(* LS Electric XG5000 project: PLC_Study *)
(* PLC LSPLC *)
(* module base 0 slot 0: 입력 모듈:XGI-D21A (DC 24V 입력, 8점 (전류소스/싱크입력)) *)
(* module base 0 slot 1: 출력 모듈:XGQ-RY1A (릴레이 출력, 8점 (2A용, 단독 COM.)) *)

(* Comments on direct variables
%QX0.1.0	출력
%QX0.1.2	출력
%IX0.0.3	스위치
*)

PROGRAM NewProgram (* task: 스캔 프로그램 *)

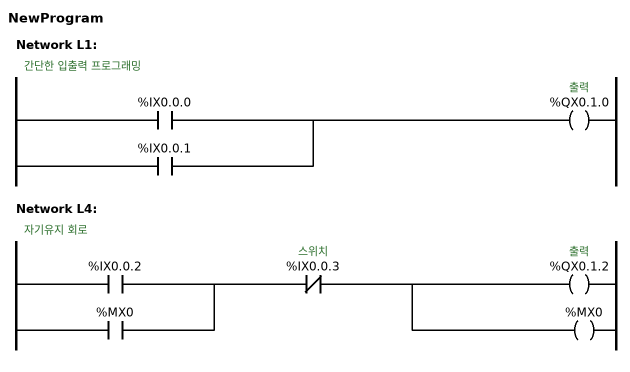
(* 간단한 입출력 프로그래밍 *)
(* Rung L1 *)
%QX0.1.0 := %IX0.0.0 OR %IX0.0.1;
(* 자기유지 회로 *)
(* Rung L4 *)
%QX0.1.2 := (%IX0.0.2 OR %MX0) AND NOT %IX0.0.3;
%MX0 := (%IX0.0.2 OR %MX0) AND NOT %IX0.0.3;
END_PROGRAM